// TIA Portal project "e058002v15" (V14)

(* hardware
DEVICE "S7-1200 station_1"  SIMATIC 1200-Station
   slot 0: "Rack S7-1200"  Rack  V1.0
   slot 1: "PLC_1"  CPU 1212C DC/DC/DC  6ES7 212-1AE31-0XB0  V3.0
   slot 2: "DI 8x24VDC/DQ 8xRelay_1"  SM 1223 DI8/DQ8 x relay  6ES7 223-1PH32-0XB0  V2.0
DEVICE "U9.3"  KTP600 Basic mono PN
   slot 0: "HMI"  HMI  6AV6 647-0AB11-3AX0  12.0.0.0
   slot 1: "HMI_RT_2"  KTP600 Basic mono PN  6AV6 647-0AB11-3AX0  12.0.0.0
   slot 5: "U9.3._CP_1"  Interfaz PROFINET
      slot 1: "Interfaz PROFINET_1"  Interfaz PROFINET
         slot 1: "Port_1"  Port
*)

// ===== PLC "PLC_1"  CPU 1212C DC/DC/DC =====

VAR_GLOBAL   // PLC tag table "Tabla de variables estándar"
   "System_Byte" AT %MB2 : Byte;
   "FirstScan" AT %M2.0 : Bool;
   "DiagStatusUpdate" AT %M2.1 : Bool;
   "AlwaysTRUE" AT %M2.2 : Bool;
   "AlwaysFALSE" AT %M2.3 : Bool;
   "Cuenta_Actual" AT %MW12 : Int;
   "PV_Cuenta_Rech" AT %MW14 : Int;
   "Reset_Cuenta" AT %M3.0 : Bool;
   "Aux_Ala_Enc" AT %MD220 : DInt;
   "Tag_1" AT %M231.0 : Bool;
   "Flanco falla de encoder" AT %M232.0 : Bool;
   "Tag_2" AT %M233.0 : Bool;
   "Tag_3" AT %M232.1 : Bool;
   "Flc_Ala_Encoder" AT %M234.0 : Bool;
   "Tag_4" AT %M231.2 : Bool;
   "Aux_Ala_Enc2" AT %MD224 : DInt;
   "Aux_Ala_Enc3" AT %MD240 : DInt;
   "Flc_FallaxCuentas" AT %M234.1 : Bool;
END_VAR

VAR_GLOBAL   // PLC tag table "00_Entradas"
   "iSns_PresenciaTapa" AT %I0.3 : Bool;   // S5.3 Sensor Presencia de Tapa
   "iSns_PresenciaBotella" AT %I0.2 : Bool;   // S5.4 Sensor Presencia de Botella
   "iCont_Encóder" AT %ID1000 : DInt;   // Valor Contador Encóder
   "reserva(1)" AT %I0.7 : Bool;   // Parada de emergencia caja mecanica
   "iPulsadorInicio" AT %I1.1 : Bool;   // Pulsador Inicio en caja mecanica.
   "iPulsadorParada" AT %I1.0 : Bool;   // Pulsador de parada en caja mecanica.
   "reserva" AT %I0.5 : Bool;   // Parada de emergencia en caja gris.
   "iSns_FuerzaDedos" AT %I1.2 : Bool;   // Sensor de fuerza de los dedos
END_VAR

VAR_GLOBAL   // PLC tag table "01_Salidas"
   "oRly_Pateador" AT %Q0.0 : Bool;   // R1 - Pateador
   "oRly_Embrague" AT %Q0.2 : Bool;   // R3 - Embrague
   "oLuzIndicadora" AT %Q0.4 : Bool;   // Luz indicadora de estado automatico/manual
END_VAR

VAR_GLOBAL   // PLC tag table "02_General"
   "SiempreEn_0" AT %M0.0 : Bool;   // Este Bit Siempre está en 0
   "SiempreEn_1" AT %M0.1 : Bool;   // Este Bit Siempre está en 1
   "Reset_Contador" AT %M0.2 : Bool;   // Señal para reset de contador
   "Modo" AT %M0.3 : Bool;   // Modo de funcionamiento- 0 : Parado 1: Automático
   "ParadaMaxBotRecha" AT %M0.4 : Bool;   // Parada Por Máxima cantidad de botellas rechazadas.
   "Falla_ParadaDeLinea" AT %M0.5 : Bool;   // Parada de linea por alguna falla.
   "mCont_Encoder_Anterior" AT %MD50 : DInt;
   "xFNPul_Parada" AT %M0.6 : Bool;
END_VAR

VAR_GLOBAL   // PLC tag table "03_Pateador"
   "PresenciaDeBotella" AT %M1.0 : Bool;   // Marca que indica precencia de botella.
   "PrecenciaDeBot_Y_Tapa" AT %M1.1 : Bool;   // Marca que indica precencia de tapa.
   "Botella_Sin_Tapa" AT %M1.2 : Bool;   // Marca que indica botella sin tapa
   "Ant_Botella_Sin_Tapa" AT %M1.3 : Bool;   // Valor anterior de marca que indica botella sin tapa.
   "Ord_Patear" AT %M1.4 : Bool;   // Orden para patear
   "Ant_Ord_Patear" AT %M1.5 : Bool;   // Valor anterior de orden para patear
   "Ant1_Ord_Patear" AT %M1.6 : Bool;
END_VAR

VAR_GLOBAL   // PLC tag table "05_Auxiliares"
   "AuxiliarSuma" AT %MD100 : DInt;
   "Auxiliar_1" AT %M104.0 : Bool;
   "Auxiliar_2" AT %M104.1 : Bool;
   "Auxiliar_3" AT %M104.2 : Bool;
   "Auxiliar_4" AT %M104.3 : Bool;
   "Auxiliar_5" AT %M104.4 : Bool;
   "Auxiliar_6" AT %M104.5 : Bool;
   "Auxiliar_7" AT %M104.6 : Bool;
   "Auxiliar_8" AT %M104.7 : Bool;
   "DWordTemp" AT %MD106 : DInt;
END_VAR

VAR_GLOBAL   // PLC tag table "06_Flancos"
   "fp_iSns_PresenciaTapa" AT %M10.0 : Bool;
   "fn_iSns_PresenciaTapa" AT %M10.1 : Bool;
   "fp_iSns_PresenciaBotella" AT %M10.2 : Bool;
   "fn_iSns_PresenciaBotella" AT %M10.3 : Bool;
END_VAR

VAR_GLOBAL   // PLC tag table "10_Simulacion"
   "sim_iSnsBotella" AT %M200.0 : Bool;
   "sim_iSnsTapa" AT %M200.1 : Bool;
   "sim_iPulInicio" AT %M200.2 : Bool;
   "sim_auxLoopEncoder" AT %M200.3 : Bool;
   "sim_auxFNLoop" AT %M200.4 : Bool;
END_VAR

DATA_BLOCK "100_Receta_Actual"   // DB1
TITLE = Datos Botellas
{ S7_Optimized_Access := 'TRUE' }
VERSION : 0.1
// En este bloque se almacenan todos los datos realacionado a las botellas, como ser el ancho, ancho de tapa, etc.
   VAR RETAIN
      Ancho_Max_Botella : DInt := 75;
      Cuenta_Patear : DInt := 430;
      Tiempo_Pateado : Time := T#50ms;
   END_VAR
BEGIN
END_DATA_BLOCK

DATA_BLOCK "102_Datos"   // DB2
{ S7_Optimized_Access := 'TRUE' }
VERSION : 0.1
   VAR
      Encoder_MaxCuenta : DInt := 1000000;   // Maxima cuenta del contador.
      Encoder_ValorActual : DInt;   // Variable donde alamceno valor de contador.
      Encoder_CuentaPatear : DInt;   // Valor de encoder que debe patear.
      Encoder_ValorFinBotella : DInt;   // Variable auxiliar para calculo de valor relativo del contador, sin reseteo
      NumMaxBotARechazar : Int;   // Numero maximo de botellas a rechazar, si pasa este numero genera una parada de linea.
      IndiceMaxBotARechazar : Int;   // Numero maximo del indice para rechazar botellas.
   END_VAR
BEGIN
END_DATA_BLOCK

DATA_BLOCK "101_Arreglo"   // DB4
TITLE = Arreglos
{ S7_Optimized_Access := 'TRUE' }
VERSION : 0.1
// Este bloque contiene los arreglos que se utilizan para la logica de cuenta para patear.
   VAR
      Arr_Cuenta_Patear : Array[0..9] of DInt;
      Indice : Int;
   END_VAR
BEGIN
END_DATA_BLOCK

DATA_BLOCK "103_Medición"   // DB6
{ S7_Optimized_Access := 'TRUE' }
VERSION : 0.1
   VAR
      AnchoBotellaMedicion : DInt;   // Medicion de ancho de botella
      ContadorMedicionInicio : DInt;   // Valor contador cuando ingresa botella
      ContadorMedicionFin : DInt;   // Valor contador cuando sale botella
      MedicionActivada : Bool;
      BotellaPresenteMedicion : Bool;
      MedicionRealizada : Bool;
   END_VAR
BEGIN
END_DATA_BLOCK

DATA_BLOCK "104_HMI_a_PLC"   // DB7
{ S7_Optimized_Access := 'TRUE' }
VERSION : 0.1
   VAR
      Reset : Bool;
      AnchoBotella : DInt := 75;
      CantidadPulsosPatear : DInt := 430;
      Tiempo_Pateado : Time := T#50ms;
      Cuenta_Actual : DInt;
   END_VAR
BEGIN
END_DATA_BLOCK

// folder: Alarma

DATA_BLOCK "ALA_PRE"   // DB70
{ S7_Optimized_Access := 'FALSE' }
VERSION : 0.1
   VAR
      Falla_09 : Bool;
      Falla_10 : Bool;
      Falla_11 : Bool;
      Falla_12 : Bool;
      Falla_13 : Bool;
      Falla_14 : Bool;
      Falla_15 : Bool;
      Falla_16 : Bool;
      Falla_01 : Bool;
      Falla_02 : Bool;
      Falla_03 : Bool;
      Falla_04 : Bool;
      Falla_05 : Bool;
      Falla_06 : Bool;
      Falla_07 : Bool;
      Falla_08 : Bool;
      Falla_25 : Bool;
      Falla_26 : Bool;
      Falla_27 : Bool;
      Falla_28 : Bool;
      Falla_29 : Bool;
      Falla_30 : Bool;
      Falla_31 : Bool;
      Falla_32 : Bool;
      Falla_17 : Bool;
      Falla_18 : Bool;
      Falla_19 : Bool;
      Falla_20 : Bool;
      Falla_21 : Bool;
      Falla_22 : Bool;
      Falla_23 : Bool;
      Falla_24 : Bool;
   END_VAR
BEGIN
END_DATA_BLOCK

DATA_BLOCK "ALA_MEM"   // DB71
{ S7_Optimized_Access := 'FALSE' }
VERSION : 0.1
   VAR
      Alarma_09 : Bool;
      Alarma_10 : Bool;
      Alarma_11 : Bool;
      Alarma_12 : Bool;
      Alarma_13 : Bool;
      Alarma_14 : Bool;
      Alarma_15 : Bool;
      Alarma_16 : Bool;
      Alarma_01 : Bool;
      Alarma_02 : Bool;
      Alarma_03 : Bool;
      Alarma_04 : Bool;
      Alarma_05 : Bool;
      Alarma_06 : Bool;
      Alarma_07 : Bool;
      Alarma_08 : Bool;
      Alarma_25 : Bool;
      Alarma_26 : Bool;
      Alarma_27 : Bool;
      Alarma_28 : Bool;
      Alarma_29 : Bool;
      Alarma_30 : Bool;
      Alarma_31 : Bool;
      Alarma_32 : Bool;
      Alarma_17 : Bool;
      Alarma_18 : Bool;
      Alarma_19 : Bool;
      Alarma_20 : Bool;
      Alarma_21 : Bool;
      Alarma_22 : Bool;
      Alarma_23 : Bool;
      Alarma_24 : Bool;
   END_VAR
BEGIN
END_DATA_BLOCK

DATA_BLOCK "ALA_REC"   // DB72
{ S7_Optimized_Access := 'FALSE' }
VERSION : 0.1
   VAR
      Ala_Rec_09 : Bool;
      Ala_Rec_10 : Bool;
      Ala_Rec_11 : Bool;
      Ala_Rec_12 : Bool;
      Ala_Rec_13 : Bool;
      Ala_Rec_14 : Bool;
      Ala_Rec_15 : Bool;
      Ala_Rec_16 : Bool;
      Ala_Rec_01 : Bool;
      Ala_Rec_02 : Bool;
      Ala_Rec_03 : Bool;
      Ala_Rec_04 : Bool;
      Ala_Rec_05 : Bool;
      Ala_Rec_06 : Bool;
      Ala_Rec_07 : Bool;
      Ala_Rec_08 : Bool;
      Ala_Rec_25 : Bool;
      Ala_Rec_26 : Bool;
      Ala_Rec_27 : Bool;
      Ala_Rec_28 : Bool;
      Ala_Rec_29 : Bool;
      Ala_Rec_30 : Bool;
      Ala_Rec_31 : Bool;
      Ala_Rec_32 : Bool;
      Ala_Rec_17 : Bool;
      Ala_Rec_18 : Bool;
      Ala_Rec_19 : Bool;
      Ala_Rec_20 : Bool;
      Ala_Rec_21 : Bool;
      Ala_Rec_22 : Bool;
      Ala_Rec_23 : Bool;
      Ala_Rec_24 : Bool;
   END_VAR
BEGIN
END_DATA_BLOCK

// folder: System blocks/Program resources

DATA_BLOCK "IEC_Timer_0_DB"   // DB5
{ S7_Optimized_Access := 'TRUE' }
AUTHOR : Simatic
FAMILY : IEC
NAME : IEC_TMR
VERSION : 1.0
// stored: InstanceOfName IEC_TIMER
"IEC_TIMER"
BEGIN
END_DATA_BLOCK

DATA_BLOCK "sim_tonLoopEncoder"   // DB8
{ S7_Optimized_Access := 'TRUE' }
AUTHOR : Simatic
FAMILY : IEC
NAME : IEC_TMR
VERSION : 1.0
// stored: InstanceOfName IEC_TIMER
"IEC_TIMER"
BEGIN
END_DATA_BLOCK

DATA_BLOCK "Temp_Parada_Cinta"   // DB9
{ S7_Optimized_Access := 'TRUE' }
AUTHOR : Simatic
FAMILY : IEC
NAME : IEC_TMR
VERSION : 1.0
// stored: InstanceOfName IEC_TIMER
"IEC_TIMER"
BEGIN
END_DATA_BLOCK

DATA_BLOCK "Bot_Rechazada"   // DB10
{ S7_Optimized_Access := 'TRUE' }
AUTHOR : Simatic
FAMILY : IEC
NAME : CNTR
VERSION : 1.0
// stored: InstanceOfName IEC_COUNTER
"IEC_COUNTER"
BEGIN
END_DATA_BLOCK

DATA_BLOCK "IEC_Timer_0_DB_1"   // DB11
{ S7_Optimized_Access := 'TRUE' }
AUTHOR : Simatic
FAMILY : IEC
NAME : IEC_TMR
VERSION : 1.0
// stored: InstanceOfName IEC_TIMER
"IEC_TIMER"
BEGIN
END_DATA_BLOCK

DATA_BLOCK "IEC_Timer_0_DB_2"   // DB12
{ S7_Optimized_Access := 'TRUE' }
AUTHOR : Simatic
FAMILY : IEC
NAME : IEC_TMR
VERSION : 1.0
// stored: InstanceOfName IEC_TIMER
"IEC_TIMER"
BEGIN
END_DATA_BLOCK

// folder: (top level)

FUNCTION "04_Pateador" : Void   // FC1, LAD
TITLE = Lógica del Pateador
{ S7_Optimized_Access := 'TRUE' }
VERSION : 0.1
// En este bloque se resuelve toda la lógica necesaria para activar el pateador.
   VAR_TEMP
      dist_Bot_a_pat : DInt;
   END_VAR
   VAR_TEMP   // added for the SCL form of the ladder/FBD networks
      _w1 : Bool;
      _w2 : Bool;
   END_VAR
BEGIN

REGION Network 1: Reset de contador.
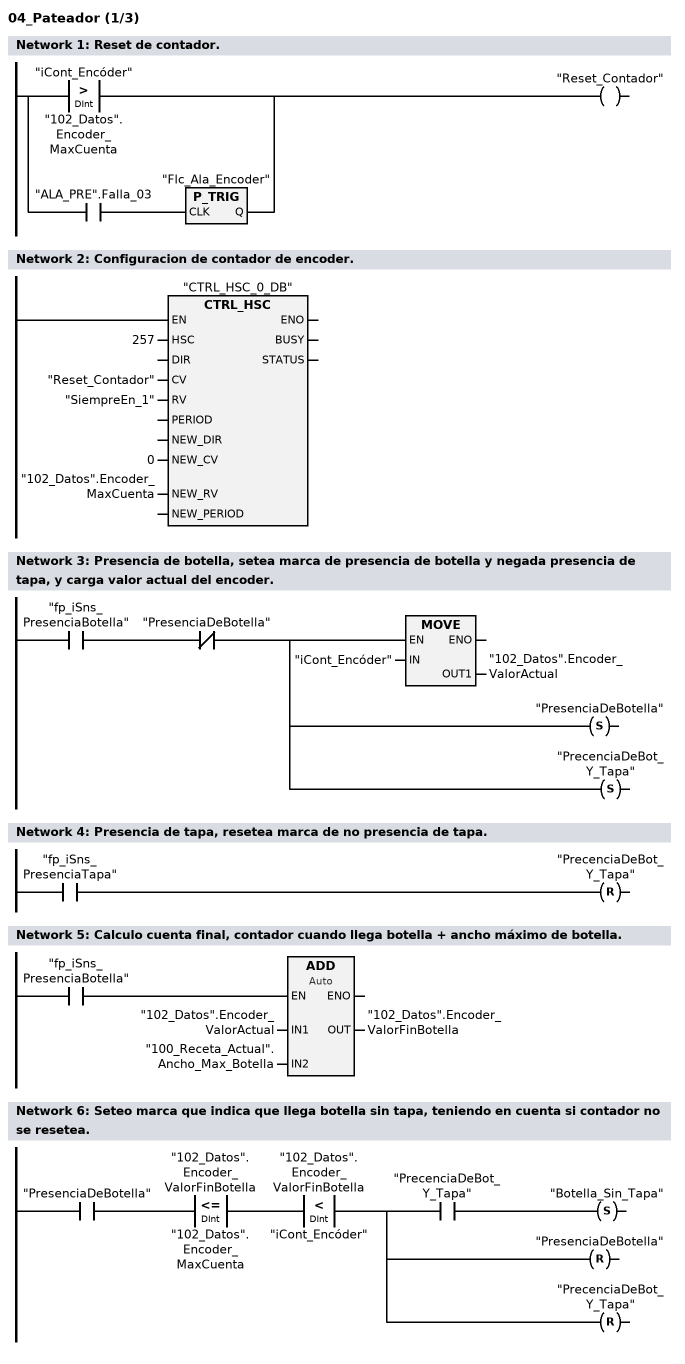
   RUNG wire#powerrail
      { S7_Templates := "SrcType := DInt" } GT_Contact(in1 := "iCont_Encóder", in2 := "102_Datos".Encoder_MaxCuenta)
      wire#w1
      Coil( "Reset_Contador" )
   END_RUNG
   RUNG wire#powerrail
      Contact( "ALA_PRE".Falla_03 )
      P_Trig( "Flc_Ala_Encoder" )
   END_RUNG wire#w1
   // the same network as SCL:
   #_w1 := "ALA_PRE".Falla_03 AND NOT "Flc_Ala_Encoder";   // rising edge
   "Flc_Ala_Encoder" := "ALA_PRE".Falla_03;
   "Reset_Contador" := ("iCont_Encóder" > "102_Datos".Encoder_MaxCuenta) OR #_w1;
END_REGION

REGION Network 2: Configuracion de contador de encoder.
   "CTRL_HSC_0_DB"(HSC := 257,   // CTRL_HSC
                   CV := "Reset_Contador",
                   RV := "SiempreEn_1",
                   NEW_CV := 0,
                   NEW_RV := "102_Datos".Encoder_MaxCuenta);
END_REGION

REGION Network 3: Presencia de botella, setea marca de presencia de botella y negada presencia de tapa, y carga valor actual del encoder.
   RUNG wire#powerrail
      Contact( "fp_iSns_PresenciaBotella" )
      I_Contact( "PresenciaDeBotella" )
      wire#w1
      { S7_GenerateENO := "TRUE" } Move(in := "iCont_Encóder", out1 => "102_Datos".Encoder_ValorActual)
   END_RUNG
   RUNG wire#w1
      S_Coil( "PresenciaDeBotella" )
   END_RUNG
   RUNG wire#w1
      S_Coil( "PrecenciaDeBot_Y_Tapa" )
   END_RUNG
   // the same network as SCL:
   IF "fp_iSns_PresenciaBotella" AND NOT "PresenciaDeBotella" THEN
       "102_Datos".Encoder_ValorActual := "iCont_Encóder";
   END_IF;
   #_w1 := "fp_iSns_PresenciaBotella" AND NOT "PresenciaDeBotella";
   IF #_w1 THEN
       "PresenciaDeBotella" := TRUE;
       "PrecenciaDeBot_Y_Tapa" := TRUE;
   END_IF;
END_REGION

REGION Network 4: Presencia de tapa, resetea marca de no presencia de tapa.
   RUNG wire#powerrail
      Contact( "fp_iSns_PresenciaTapa" )
      R_Coil( "PrecenciaDeBot_Y_Tapa" )
   END_RUNG
   // the same network as SCL:
   IF "fp_iSns_PresenciaTapa" THEN "PrecenciaDeBot_Y_Tapa" := FALSE; END_IF;
END_REGION

REGION Network 5: Calculo cuenta final, contador cuando llega botella + ancho máximo de botella.
   RUNG wire#powerrail
      Contact( "fp_iSns_PresenciaBotella" )
      { S7_GenerateENO := "TRUE" } Add(in1 := "102_Datos".Encoder_ValorActual, in2 := "100_Receta_Actual".Ancho_Max_Botella, out => "102_Datos".Encoder_ValorFinBotella)
   END_RUNG
   // the same network as SCL:
   IF "fp_iSns_PresenciaBotella" THEN
       "102_Datos".Encoder_ValorFinBotella := "102_Datos".Encoder_ValorActual + "100_Receta_Actual".Ancho_Max_Botella;
   END_IF;
END_REGION

REGION Network 6: Seteo marca que indica que llega botella sin tapa, teniendo en cuenta si contador no se resetea.
   RUNG wire#powerrail
      Contact( "PresenciaDeBotella" )
      { S7_Templates := "SrcType := DInt" } LE_Contact(in1 := "102_Datos".Encoder_ValorFinBotella, in2 := "102_Datos".Encoder_MaxCuenta)
      { S7_Templates := "SrcType := DInt" } LT_Contact(in1 := "102_Datos".Encoder_ValorFinBotella, in2 := "iCont_Encóder")
      wire#w1
      Contact( "PrecenciaDeBot_Y_Tapa" )
      S_Coil( "Botella_Sin_Tapa" )
   END_RUNG
   RUNG wire#w1
      R_Coil( "PresenciaDeBotella" )
   END_RUNG
   RUNG wire#w1
      R_Coil( "PrecenciaDeBot_Y_Tapa" )
   END_RUNG
   // the same network as SCL:
   #_w1 := "PresenciaDeBotella" AND ("102_Datos".Encoder_ValorFinBotella <= "102_Datos".Encoder_MaxCuenta) AND ("102_Datos".Encoder_ValorFinBotella < "iCont_Encóder");
   IF #_w1 AND "PrecenciaDeBot_Y_Tapa" THEN "Botella_Sin_Tapa" := TRUE; END_IF;
   IF #_w1 THEN
       "PresenciaDeBotella" := FALSE;
       "PrecenciaDeBot_Y_Tapa" := FALSE;
   END_IF;
END_REGION

REGION Network 7: Seteo marca que indica que llega botella sin tapa, teniendo en cuenta el caso que el contador se resetea.
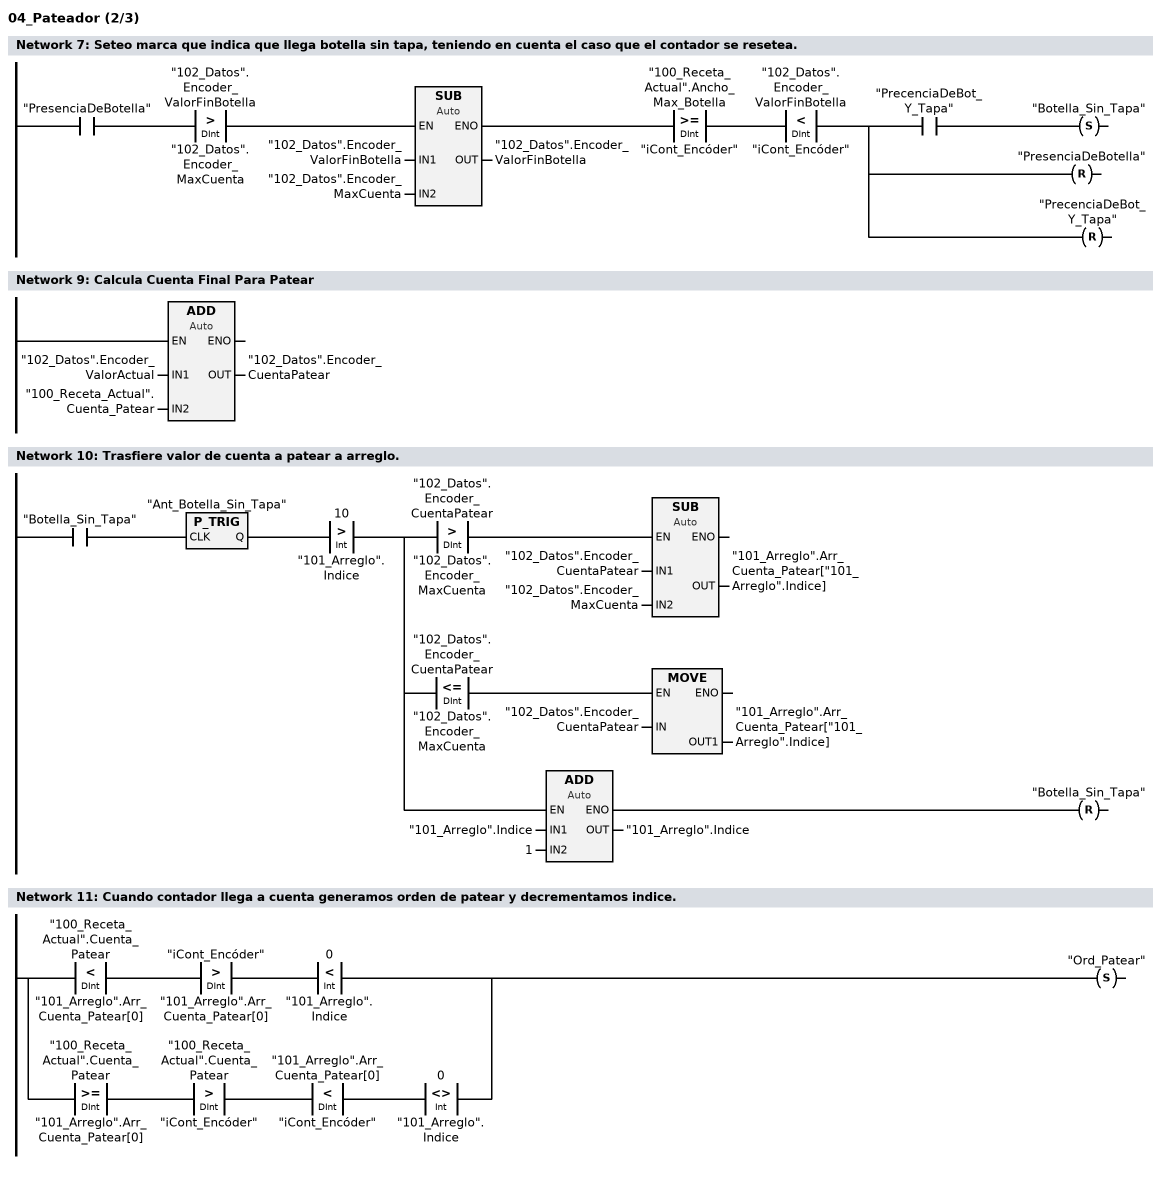
   RUNG wire#powerrail
      Contact( "PresenciaDeBotella" )
      { S7_Templates := "SrcType := DInt" } GT_Contact(in1 := "102_Datos".Encoder_ValorFinBotella, in2 := "102_Datos".Encoder_MaxCuenta)
      { S7_GenerateENO := "TRUE" } Sub(in1 := "102_Datos".Encoder_ValorFinBotella, in2 := "102_Datos".Encoder_MaxCuenta, out => "102_Datos".Encoder_ValorFinBotella)
      { S7_Templates := "SrcType := DInt" } GE_Contact(in1 := "100_Receta_Actual".Ancho_Max_Botella, in2 := "iCont_Encóder")
      { S7_Templates := "SrcType := DInt" } LT_Contact(in1 := "102_Datos".Encoder_ValorFinBotella, in2 := "iCont_Encóder")
      wire#w1
      Contact( "PrecenciaDeBot_Y_Tapa" )
      S_Coil( "Botella_Sin_Tapa" )
   END_RUNG
   RUNG wire#w1
      R_Coil( "PresenciaDeBotella" )
   END_RUNG
   RUNG wire#w1
      R_Coil( "PrecenciaDeBot_Y_Tapa" )
   END_RUNG
   // the same network as SCL:
   // ENO of a box is taken as its EN; it also drops when the box reports an error
   #_w1 := "PresenciaDeBotella" AND ("102_Datos".Encoder_ValorFinBotella > "102_Datos".Encoder_MaxCuenta);
   IF #_w1 THEN
       "102_Datos".Encoder_ValorFinBotella := "102_Datos".Encoder_ValorFinBotella - "102_Datos".Encoder_MaxCuenta;
   END_IF;
   #_w2 := #_w1 AND ("100_Receta_Actual".Ancho_Max_Botella >= "iCont_Encóder") AND ("102_Datos".Encoder_ValorFinBotella < "iCont_Encóder");
   IF #_w2 AND "PrecenciaDeBot_Y_Tapa" THEN "Botella_Sin_Tapa" := TRUE; END_IF;
   IF #_w2 THEN
       "PresenciaDeBotella" := FALSE;
       "PrecenciaDeBot_Y_Tapa" := FALSE;
   END_IF;
END_REGION

REGION Network 8: Marca que indica precencia de botella.
END_REGION

REGION Network 9: Calcula Cuenta Final Para Patear
   RUNG wire#powerrail
      { S7_GenerateENO := "TRUE" } Add(in1 := "102_Datos".Encoder_ValorActual, in2 := "100_Receta_Actual".Cuenta_Patear, out => "102_Datos".Encoder_CuentaPatear)
   END_RUNG
   // the same network as SCL:
   "102_Datos".Encoder_CuentaPatear := "102_Datos".Encoder_ValorActual + "100_Receta_Actual".Cuenta_Patear;
END_REGION

REGION Network 10: Trasfiere valor de cuenta a patear a arreglo.
   RUNG wire#powerrail
      Contact( "Botella_Sin_Tapa" )
      P_Trig( "Ant_Botella_Sin_Tapa" )
      { S7_Templates := "SrcType := Int" } GT_Contact(in1 := 10, in2 := "101_Arreglo".Indice)
      wire#w1
      { S7_Templates := "SrcType := DInt" } GT_Contact(in1 := "102_Datos".Encoder_CuentaPatear, in2 := "102_Datos".Encoder_MaxCuenta)
      { S7_GenerateENO := "TRUE" } Sub(in1 := "102_Datos".Encoder_CuentaPatear, in2 := "102_Datos".Encoder_MaxCuenta, out => "101_Arreglo".Arr_Cuenta_Patear["101_Arreglo".Indice])
   END_RUNG
   RUNG wire#w1
      { S7_Templates := "SrcType := DInt" } LE_Contact(in1 := "102_Datos".Encoder_CuentaPatear, in2 := "102_Datos".Encoder_MaxCuenta)
      { S7_GenerateENO := "TRUE" } Move(in := "102_Datos".Encoder_CuentaPatear, out1 => "101_Arreglo".Arr_Cuenta_Patear["101_Arreglo".Indice])
   END_RUNG
   RUNG wire#w1
      { S7_GenerateENO := "TRUE" } Add(in1 := "101_Arreglo".Indice, in2 := 1, out => "101_Arreglo".Indice)
      R_Coil( "Botella_Sin_Tapa" )
   END_RUNG
   // the same network as SCL:
   // ENO of a box is taken as its EN; it also drops when the box reports an error
   #_w1 := "Botella_Sin_Tapa" AND NOT "Ant_Botella_Sin_Tapa";   // rising edge
   "Ant_Botella_Sin_Tapa" := "Botella_Sin_Tapa";
   #_w2 := #_w1 AND (10 > "101_Arreglo".Indice);
   IF #_w2 AND ("102_Datos".Encoder_CuentaPatear > "102_Datos".Encoder_MaxCuenta) THEN
       "101_Arreglo".Arr_Cuenta_Patear["101_Arreglo".Indice] := "102_Datos".Encoder_CuentaPatear - "102_Datos".Encoder_MaxCuenta;
   END_IF;
   IF #_w2 AND ("102_Datos".Encoder_CuentaPatear <= "102_Datos".Encoder_MaxCuenta) THEN
       "101_Arreglo".Arr_Cuenta_Patear["101_Arreglo".Indice] := "102_Datos".Encoder_CuentaPatear;
   END_IF;
   IF #_w2 THEN
       "101_Arreglo".Indice := "101_Arreglo".Indice + 1;
       "Botella_Sin_Tapa" := FALSE;
   END_IF;
END_REGION

REGION Network 11: Cuando contador llega a cuenta generamos orden de patear y decrementamos indice.
   RUNG wire#powerrail
      { S7_Templates := "SrcType := DInt" } LT_Contact(in1 := "100_Receta_Actual".Cuenta_Patear, in2 := "101_Arreglo".Arr_Cuenta_Patear[0])
      { S7_Templates := "SrcType := DInt" } GT_Contact(in1 := "iCont_Encóder", in2 := "101_Arreglo".Arr_Cuenta_Patear[0])
      { S7_Templates := "SrcType := Int" } LT_Contact(in1 := 0, in2 := "101_Arreglo".Indice)
      wire#w1
      S_Coil( "Ord_Patear" )
   END_RUNG
   RUNG wire#powerrail
      { S7_Templates := "SrcType := DInt" } GE_Contact(in1 := "100_Receta_Actual".Cuenta_Patear, in2 := "101_Arreglo".Arr_Cuenta_Patear[0])
      { S7_Templates := "SrcType := DInt" } GT_Contact(in1 := "100_Receta_Actual".Cuenta_Patear, in2 := "iCont_Encóder")
      { S7_Templates := "SrcType := DInt" } LT_Contact(in1 := "101_Arreglo".Arr_Cuenta_Patear[0], in2 := "iCont_Encóder")
      { S7_Templates := "SrcType := Int" } NE_Contact(in1 := 0, in2 := "101_Arreglo".Indice)
   END_RUNG wire#w1
   // the same network as SCL:
   IF (("100_Receta_Actual".Cuenta_Patear < "101_Arreglo".Arr_Cuenta_Patear[0]) AND ("iCont_Encóder" > "101_Arreglo".Arr_Cuenta_Patear[0]) AND (0 < "101_Arreglo".Indice)) OR (("100_Receta_Actual".Cuenta_Patear >= "101_Arreglo".Arr_Cuenta_Patear[0]) AND ("100_Receta_Actual".Cuenta_Patear > "iCont_Encóder") AND ("101_Arreglo".Arr_Cuenta_Patear[0] < "iCont_Encóder") AND (0 <> "101_Arreglo".Indice)) THEN
       "Ord_Patear" := TRUE;
   END_IF;
END_REGION

REGION Network 12: Correr Arreglo En una Valor de 1 a 0 y activo salida por un timepo determinado y decrementa indice
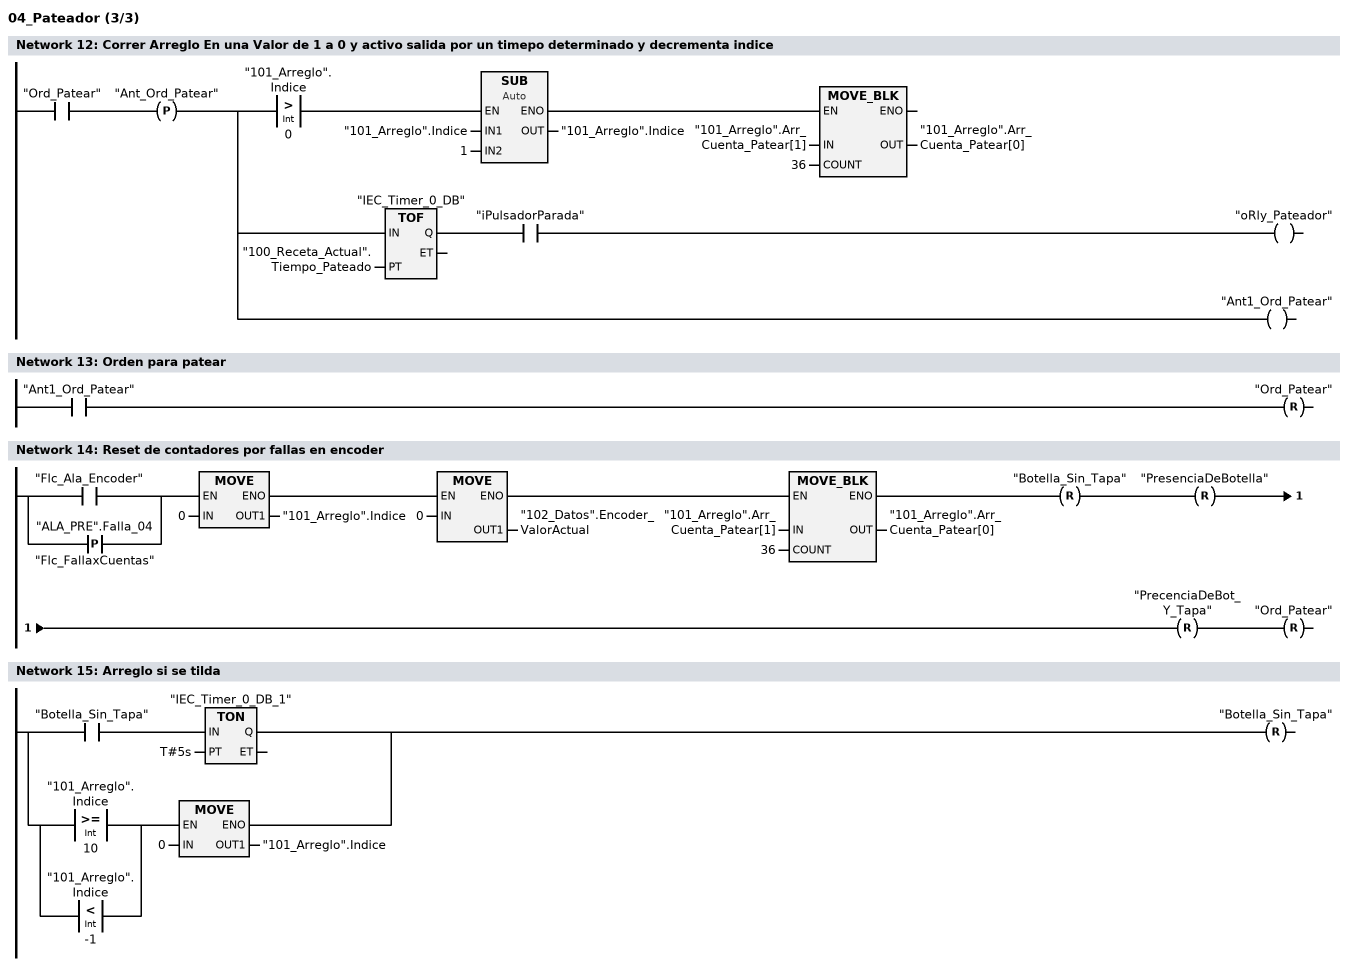
   // ENO of a box is taken as its EN; it also drops when the box reports an error
   #_w1 := "Ord_Patear" AND NOT "Ant_Ord_Patear";   // rising edge
   "Ant_Ord_Patear" := "Ord_Patear";
   #_w2 := #_w1 AND ("101_Arreglo".Indice > 0);
   IF #_w2 THEN
       "101_Arreglo".Indice := "101_Arreglo".Indice - 1;
       MOVE_BLK(IN := "101_Arreglo".Arr_Cuenta_Patear[1], COUNT := 36, OUT => "101_Arreglo".Arr_Cuenta_Patear[0]);
   END_IF;
   "IEC_Timer_0_DB".TOF(IN := #_w1, PT := "100_Receta_Actual".Tiempo_Pateado);
   "oRly_Pateador" := "IEC_Timer_0_DB".Q AND "iPulsadorParada";
   "Ant1_Ord_Patear" := #_w1;
END_REGION

REGION Network 13: Orden para patear
   RUNG wire#powerrail
      Contact( "Ant1_Ord_Patear" )
      R_Coil( "Ord_Patear" )
   END_RUNG
   // the same network as SCL:
   IF "Ant1_Ord_Patear" THEN "Ord_Patear" := FALSE; END_IF;
END_REGION

REGION Network 14: Reset de contadores por fallas en encoder
   // ENO of a box is taken as its EN; it also drops when the box reports an error
   #_w1 := "ALA_PRE".Falla_04 AND NOT "Flc_FallaxCuentas";   // rising edge of "ALA_PRE".Falla_04
   "Flc_FallaxCuentas" := "ALA_PRE".Falla_04;
   IF "Flc_Ala_Encoder" OR #_w1 THEN
       "101_Arreglo".Indice := 0;
       "102_Datos".Encoder_ValorActual := 0;
   END_IF;
   #_w2 := "Flc_Ala_Encoder" OR #_w1;
   IF #_w2 THEN
       MOVE_BLK(IN := "101_Arreglo".Arr_Cuenta_Patear[1], COUNT := 36, OUT => "101_Arreglo".Arr_Cuenta_Patear[0]);
       "Botella_Sin_Tapa" := FALSE;
       "PresenciaDeBotella" := FALSE;
       "PrecenciaDeBot_Y_Tapa" := FALSE;
       "Ord_Patear" := FALSE;
   END_IF;
END_REGION

REGION Network 15: Arreglo si se tilda
   // ENO of a box is taken as its EN; it also drops when the box reports an error
   "IEC_Timer_0_DB_1".TON(IN := "Botella_Sin_Tapa", PT := T#5s);
   #_w1 := ("101_Arreglo".Indice >= 10) OR ("101_Arreglo".Indice < (-1));
   IF #_w1 THEN "101_Arreglo".Indice := 0; END_IF;
   IF "IEC_Timer_0_DB_1".Q OR #_w1 THEN "Botella_Sin_Tapa" := FALSE; END_IF;
END_REGION
END_FUNCTION

FUNCTION "03_Medicion" : Void   // FC2, LAD
TITLE = Medicion
{ S7_Optimized_Access := 'TRUE' }
VERSION : 0.1
// En este bloque realizamos la medicion del ancho de la botella.
   VAR_TEMP   // added for the SCL form of the ladder/FBD networks
      _w1 : Bool;
   END_VAR
BEGIN

REGION Network 1: Guardamos valor de contador cuando llega botella.
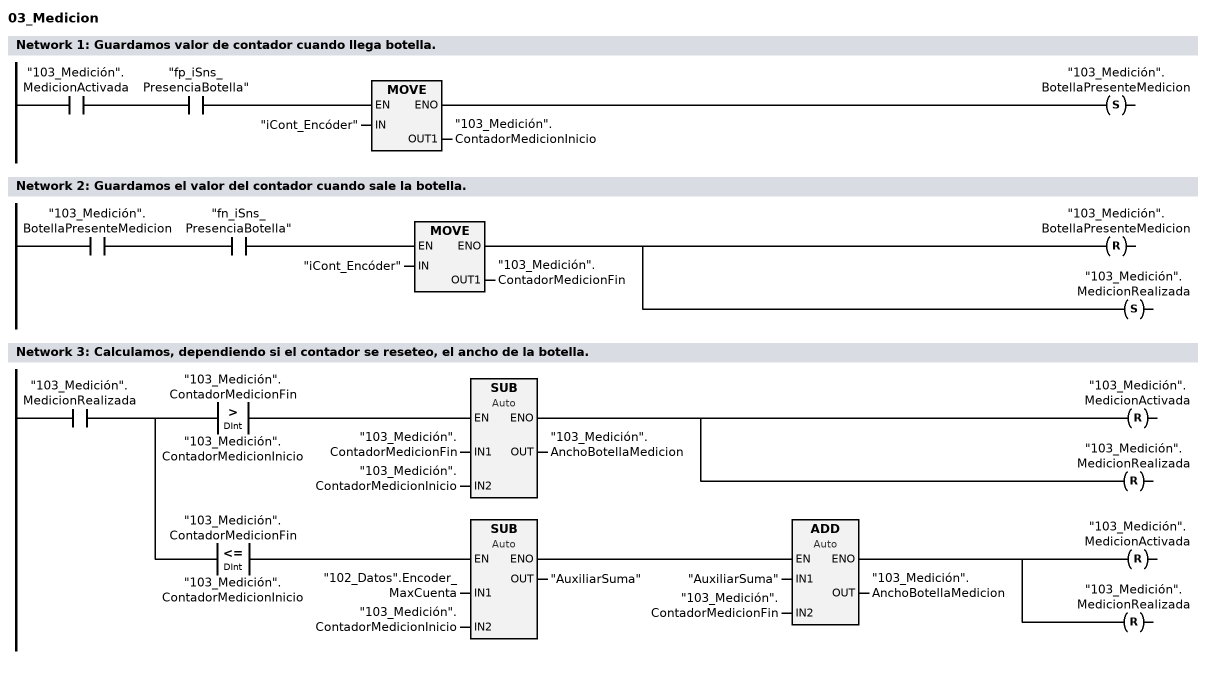
   RUNG wire#powerrail
      Contact( "103_Medición".MedicionActivada )
      Contact( "fp_iSns_PresenciaBotella" )
      { S7_GenerateENO := "TRUE" } Move(in := "iCont_Encóder", out1 => "103_Medición".ContadorMedicionInicio)
      S_Coil( "103_Medición".BotellaPresenteMedicion )
   END_RUNG
   // the same network as SCL:
   // ENO of a box is taken as its EN; it also drops when the box reports an error
   IF "103_Medición".MedicionActivada AND "fp_iSns_PresenciaBotella" THEN
       "103_Medición".ContadorMedicionInicio := "iCont_Encóder";
       "103_Medición".BotellaPresenteMedicion := TRUE;
   END_IF;
END_REGION

REGION Network 2: Guardamos el valor del contador cuando sale la botella.
   RUNG wire#powerrail
      Contact( "103_Medición".BotellaPresenteMedicion )
      Contact( "fn_iSns_PresenciaBotella" )
      { S7_GenerateENO := "TRUE" } Move(in := "iCont_Encóder", out1 => "103_Medición".ContadorMedicionFin)
      wire#w1
      R_Coil( "103_Medición".BotellaPresenteMedicion )
   END_RUNG
   RUNG wire#w1
      S_Coil( "103_Medición".MedicionRealizada )
   END_RUNG
   // the same network as SCL:
   // ENO of a box is taken as its EN; it also drops when the box reports an error
   IF "103_Medición".BotellaPresenteMedicion AND "fn_iSns_PresenciaBotella" THEN
       "103_Medición".ContadorMedicionFin := "iCont_Encóder";
   END_IF;
   #_w1 := "103_Medición".BotellaPresenteMedicion AND "fn_iSns_PresenciaBotella";
   IF #_w1 THEN
       "103_Medición".BotellaPresenteMedicion := FALSE;
       "103_Medición".MedicionRealizada := TRUE;
   END_IF;
END_REGION

REGION Network 3: Calculamos, dependiendo si el contador se reseteo, el ancho de la botella.
   RUNG wire#powerrail
      Contact( "103_Medición".MedicionRealizada )
      wire#w1
      { S7_Templates := "SrcType := DInt" } GT_Contact(in1 := "103_Medición".ContadorMedicionFin, in2 := "103_Medición".ContadorMedicionInicio)
      { S7_GenerateENO := "TRUE" } Sub(in1 := "103_Medición".ContadorMedicionFin, in2 := "103_Medición".ContadorMedicionInicio, out => "103_Medición".AnchoBotellaMedicion)
      wire#w2
      R_Coil( "103_Medición".MedicionActivada )
   END_RUNG
   RUNG wire#w2
      R_Coil( "103_Medición".MedicionRealizada )
   END_RUNG
   RUNG wire#w1
      { S7_Templates := "SrcType := DInt" } LE_Contact(in1 := "103_Medición".ContadorMedicionFin, in2 := "103_Medición".ContadorMedicionInicio)
      { S7_GenerateENO := "TRUE" } Sub(in1 := "102_Datos".Encoder_MaxCuenta, in2 := "103_Medición".ContadorMedicionInicio, out => "AuxiliarSuma")
      { S7_GenerateENO := "TRUE" } Add(in1 := "AuxiliarSuma", in2 := "103_Medición".ContadorMedicionFin, out => "103_Medición".AnchoBotellaMedicion)
      wire#w3
      R_Coil( "103_Medición".MedicionActivada )
   END_RUNG
   RUNG wire#w3
      R_Coil( "103_Medición".MedicionRealizada )
   END_RUNG
   // the same network as SCL:
   // ENO of a box is taken as its EN; it also drops when the box reports an error
   IF "103_Medición".MedicionRealizada AND ("103_Medición".ContadorMedicionFin > "103_Medición".ContadorMedicionInicio) THEN
       "103_Medición".AnchoBotellaMedicion := "103_Medición".ContadorMedicionFin - "103_Medición".ContadorMedicionInicio;
       "103_Medición".MedicionActivada := FALSE;
   END_IF;
   #_w1 := "103_Medición".MedicionRealizada;
   IF "103_Medición".MedicionRealizada AND ("103_Medición".ContadorMedicionFin > "103_Medición".ContadorMedicionInicio) THEN
       "103_Medición".MedicionRealizada := FALSE;
   END_IF;
   IF #_w1 AND ("103_Medición".ContadorMedicionFin <= "103_Medición".ContadorMedicionInicio) THEN
       "AuxiliarSuma" := "102_Datos".Encoder_MaxCuenta - "103_Medición".ContadorMedicionInicio;
       "103_Medición".AnchoBotellaMedicion := "AuxiliarSuma" + "103_Medición".ContadorMedicionFin;
       "103_Medición".MedicionActivada := FALSE;
       "103_Medición".MedicionRealizada := FALSE;
   END_IF;
END_REGION
END_FUNCTION

FUNCTION "00_Alarmas" : Void   // FC3, LAD
{ S7_Optimized_Access := 'TRUE' }
VERSION : 0.1
   VAR_TEMP
      dist_Bot_a_pat : DInt;
   END_VAR
   VAR_TEMP   // added for the SCL form of the ladder/FBD networks
      _w1 : Bool;
   END_VAR
BEGIN

REGION Network 1: Parada manual. Emergencia o Stop del embrague del pateador.
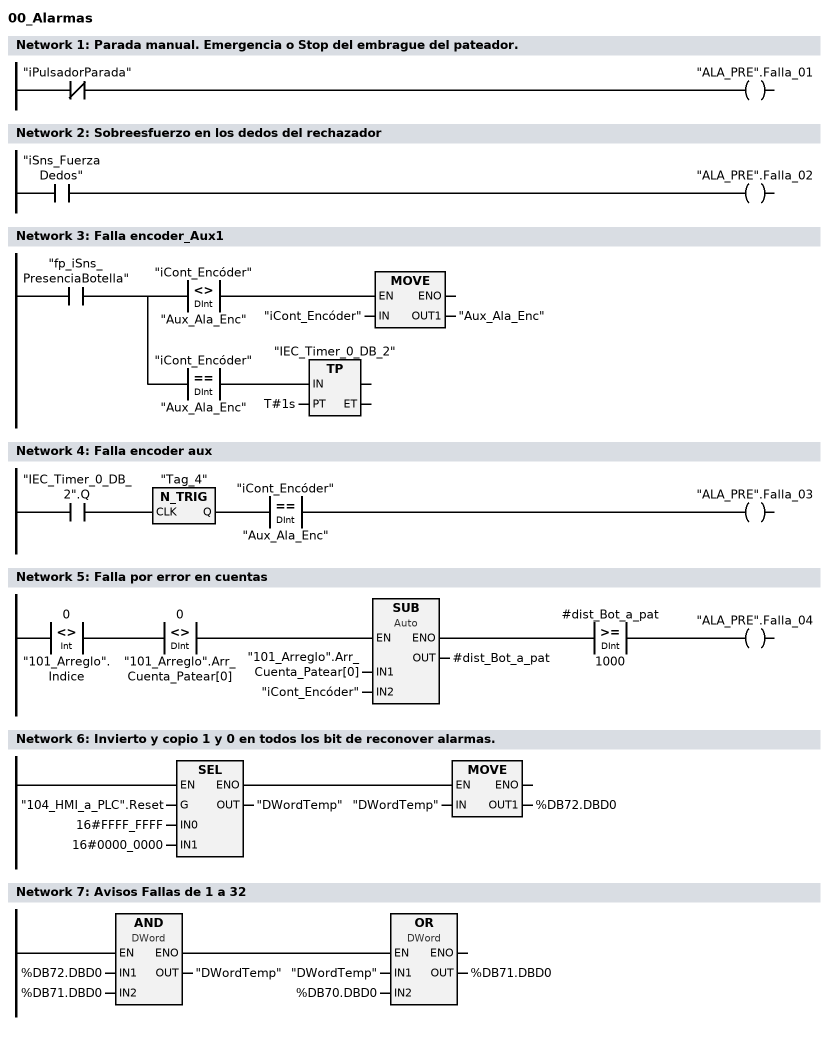
   RUNG wire#powerrail
      I_Contact( "iPulsadorParada" )
      Coil( "ALA_PRE".Falla_01 )
   END_RUNG
   // the same network as SCL:
   "ALA_PRE".Falla_01 := NOT "iPulsadorParada";
END_REGION

REGION Network 2: Sobreesfuerzo en los dedos del rechazador
   RUNG wire#powerrail
      Contact( "iSns_FuerzaDedos" )
      Coil( "ALA_PRE".Falla_02 )
   END_RUNG
   // the same network as SCL:
   "ALA_PRE".Falla_02 := "iSns_FuerzaDedos";
END_REGION

REGION Network 3: Falla encoder_Aux1
   IF "fp_iSns_PresenciaBotella" AND ("iCont_Encóder" <> "Aux_Ala_Enc") THEN
       "Aux_Ala_Enc" := "iCont_Encóder";
   END_IF;
   "IEC_Timer_0_DB_2".TP(IN := "fp_iSns_PresenciaBotella" AND ("iCont_Encóder" = "Aux_Ala_Enc"), PT := T#1s);
END_REGION

REGION Network 4: Falla encoder aux
   RUNG wire#powerrail
      Contact( "IEC_Timer_0_DB_2".Q )
      N_Trig( "Tag_4" )
      { S7_Templates := "SrcType := DInt" } EQ_Contact(in1 := "iCont_Encóder", in2 := "Aux_Ala_Enc")
      Coil( "ALA_PRE".Falla_03 )
   END_RUNG
   // the same network as SCL:
   #_w1 := NOT "IEC_Timer_0_DB_2".Q AND "Tag_4";   // falling edge
   "Tag_4" := "IEC_Timer_0_DB_2".Q;
   "ALA_PRE".Falla_03 := #_w1 AND ("iCont_Encóder" = "Aux_Ala_Enc");
END_REGION

REGION Network 5: Falla por error en cuentas
   RUNG wire#powerrail
      { S7_Templates := "SrcType := Int" } NE_Contact(in1 := 0, in2 := "101_Arreglo".Indice)
      { S7_Templates := "SrcType := DInt" } NE_Contact(in1 := 0, in2 := "101_Arreglo".Arr_Cuenta_Patear[0])
      { S7_GenerateENO := "TRUE" } Sub(in1 := "101_Arreglo".Arr_Cuenta_Patear[0], in2 := "iCont_Encóder", out => #dist_Bot_a_pat)
      { S7_Templates := "SrcType := DInt" } GE_Contact(in1 := #dist_Bot_a_pat, in2 := 1000)
      Coil( "ALA_PRE".Falla_04 )
   END_RUNG
   // the same network as SCL:
   // ENO of a box is taken as its EN; it also drops when the box reports an error
   #_w1 := (0 <> "101_Arreglo".Indice) AND (0 <> "101_Arreglo".Arr_Cuenta_Patear[0]);
   IF #_w1 THEN #dist_Bot_a_pat := "101_Arreglo".Arr_Cuenta_Patear[0] - "iCont_Encóder"; END_IF;
   "ALA_PRE".Falla_04 := #_w1 AND (#dist_Bot_a_pat >= 1000);
END_REGION

REGION Network 6: Invierto y copio 1 y 0 en todos los bit de reconover alarmas.
   // ENO of a box is taken as its EN; it also drops when the box reports an error
   "DWordTemp" := SEL(G := "104_HMI_a_PLC".Reset, IN0 := 16#FFFF_FFFF, IN1 := 16#0000_0000);
   %DB72.DBD0 := "DWordTemp";
END_REGION

REGION Network 7: Avisos Fallas de 1 a 32
   // no checked SCL form for this network; see the picture
END_REGION
END_FUNCTION

FUNCTION "01_General" : Void   // FC4, LAD
{ S7_Optimized_Access := 'TRUE' }
VERSION : 0.1
BEGIN

REGION Network 1: Set modo automatico
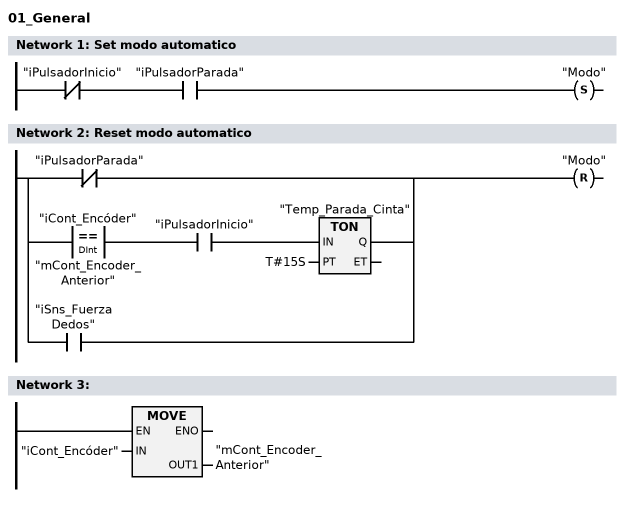
   RUNG wire#powerrail
      I_Contact( "iPulsadorInicio" )
      Contact( "iPulsadorParada" )
      S_Coil( "Modo" )
   END_RUNG
   // the same network as SCL:
   IF NOT "iPulsadorInicio" AND "iPulsadorParada" THEN "Modo" := TRUE; END_IF;
END_REGION

REGION Network 2: Reset modo automatico
   "Temp_Parada_Cinta".TON(IN := ("iCont_Encóder" = "mCont_Encoder_Anterior") AND "iPulsadorInicio",
                           PT := T#15S);
   IF NOT "iPulsadorParada" OR "Temp_Parada_Cinta".Q OR "iSns_FuerzaDedos" THEN "Modo" := FALSE; END_IF;
END_REGION

REGION Network 3
   RUNG wire#powerrail
      { S7_GenerateENO := "TRUE" } Move(in := "iCont_Encóder", out1 => "mCont_Encoder_Anterior")
   END_RUNG
   // the same network as SCL:
   "mCont_Encoder_Anterior" := "iCont_Encóder";
END_REGION
END_FUNCTION

FUNCTION "06_Salidas" : Void   // FC5, LAD
{ S7_Optimized_Access := 'TRUE' }
VERSION : 0.1
BEGIN

REGION Network 1: R3 - Embrague
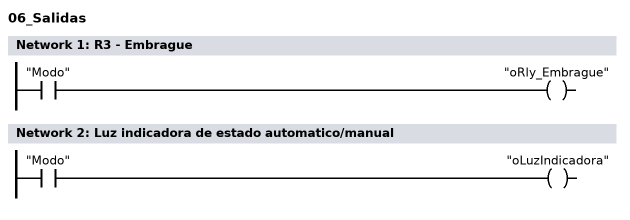
   RUNG wire#powerrail
      Contact( "Modo" )
      Coil( "oRly_Embrague" )
   END_RUNG
   // the same network as SCL:
   "oRly_Embrague" := "Modo";
END_REGION

REGION Network 2: Luz indicadora de estado automatico/manual
   RUNG wire#powerrail
      Contact( "Modo" )
      Coil( "oLuzIndicadora" )
   END_RUNG
   // the same network as SCL:
   "oLuzIndicadora" := "Modo";
END_REGION
END_FUNCTION

FUNCTION "02_Flancos" : Void   // FC6, LAD
{ S7_Optimized_Access := 'TRUE' }
VERSION : 0.1
   VAR_TEMP   // added for the SCL form of the ladder/FBD networks
      _w1 : Bool;
   END_VAR
BEGIN

REGION Network 1: Flanco Positivo Sensor Presencia de botella.
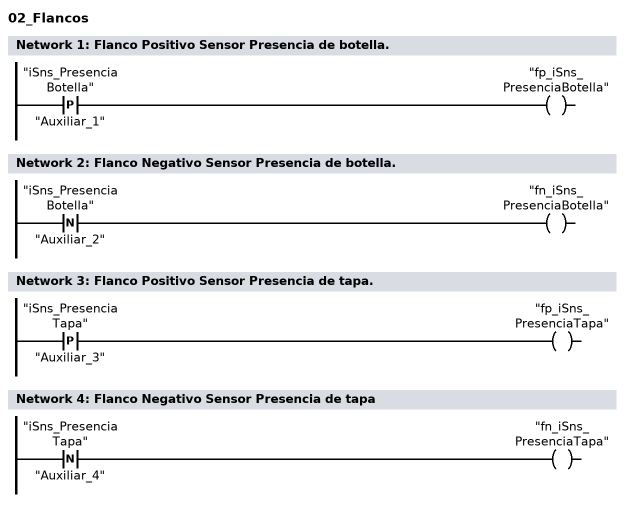
   RUNG wire#powerrail
      P_Contact(operand := "iSns_PresenciaBotella", bit := "Auxiliar_1")
      Coil( "fp_iSns_PresenciaBotella" )
   END_RUNG
   // the same network as SCL:
   #_w1 := "iSns_PresenciaBotella" AND NOT "Auxiliar_1";   // rising edge of "iSns_PresenciaBotella"
   "Auxiliar_1" := "iSns_PresenciaBotella";
   "fp_iSns_PresenciaBotella" := #_w1;
END_REGION

REGION Network 2: Flanco Negativo Sensor Presencia de botella.
   RUNG wire#powerrail
      N_Contact(operand := "iSns_PresenciaBotella", bit := "Auxiliar_2")
      Coil( "fn_iSns_PresenciaBotella" )
   END_RUNG
   // the same network as SCL:
   #_w1 := NOT "iSns_PresenciaBotella" AND "Auxiliar_2";   // falling edge of "iSns_PresenciaBotella"
   "Auxiliar_2" := "iSns_PresenciaBotella";
   "fn_iSns_PresenciaBotella" := #_w1;
END_REGION

REGION Network 3: Flanco Positivo Sensor Presencia de tapa.
   RUNG wire#powerrail
      P_Contact(operand := "iSns_PresenciaTapa", bit := "Auxiliar_3")
      Coil( "fp_iSns_PresenciaTapa" )
   END_RUNG
   // the same network as SCL:
   #_w1 := "iSns_PresenciaTapa" AND NOT "Auxiliar_3";   // rising edge of "iSns_PresenciaTapa"
   "Auxiliar_3" := "iSns_PresenciaTapa";
   "fp_iSns_PresenciaTapa" := #_w1;
END_REGION

REGION Network 4: Flanco Negativo Sensor Presencia de tapa
   RUNG wire#powerrail
      N_Contact(operand := "iSns_PresenciaTapa", bit := "Auxiliar_4")
      Coil( "fn_iSns_PresenciaTapa" )
   END_RUNG
   // the same network as SCL:
   #_w1 := NOT "iSns_PresenciaTapa" AND "Auxiliar_4";   // falling edge of "iSns_PresenciaTapa"
   "Auxiliar_4" := "iSns_PresenciaTapa";
   "fn_iSns_PresenciaTapa" := #_w1;
END_REGION
END_FUNCTION

FUNCTION "10_Simulacion" : Void   // FC7, LAD
{ S7_Optimized_Access := 'TRUE' }
VERSION : 0.1
   VAR_TEMP   // added for the SCL form of the ladder/FBD networks
      _w1 : Bool;
   END_VAR
BEGIN

REGION Network 1: Pulsador Inicio en caja mecanica.
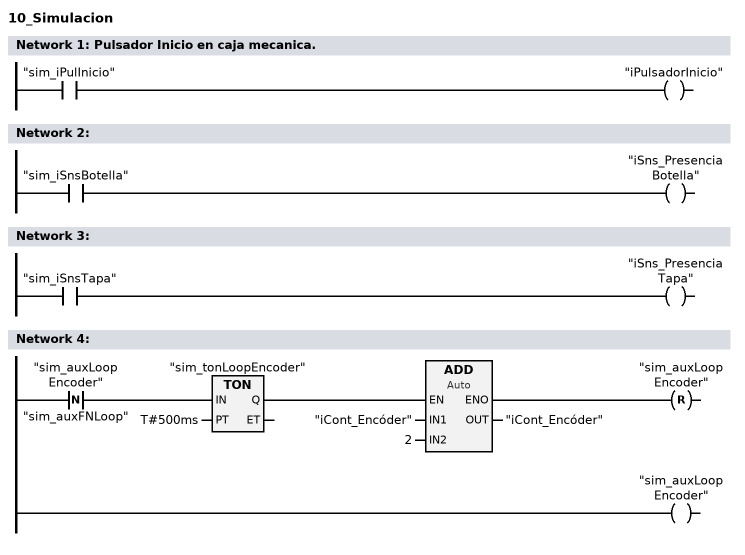
   RUNG wire#powerrail
      Contact( "sim_iPulInicio" )
      Coil( "iPulsadorInicio" )
   END_RUNG
   // the same network as SCL:
   "iPulsadorInicio" := "sim_iPulInicio";
END_REGION

REGION Network 2
   RUNG wire#powerrail
      Contact( "sim_iSnsBotella" )
      Coil( "iSns_PresenciaBotella" )
   END_RUNG
   // the same network as SCL:
   "iSns_PresenciaBotella" := "sim_iSnsBotella";
END_REGION

REGION Network 3
   RUNG wire#powerrail
      Contact( "sim_iSnsTapa" )
      Coil( "iSns_PresenciaTapa" )
   END_RUNG
   // the same network as SCL:
   "iSns_PresenciaTapa" := "sim_iSnsTapa";
END_REGION

REGION Network 4
   // ENO of a box is taken as its EN; it also drops when the box reports an error
   #_w1 := NOT "sim_auxLoopEncoder" AND "sim_auxFNLoop";   // falling edge of "sim_auxLoopEncoder"
   "sim_auxFNLoop" := "sim_auxLoopEncoder";
   "sim_tonLoopEncoder".TON(IN := #_w1, PT := T#500ms);
   IF "sim_tonLoopEncoder".Q THEN
       "iCont_Encóder" := "iCont_Encóder" + 2;
       "sim_auxLoopEncoder" := FALSE;
   END_IF;
   "sim_auxLoopEncoder" := TRUE;
END_REGION
END_FUNCTION

FUNCTION "07_HMI" : Void   // FC9, LAD
{ S7_Optimized_Access := 'TRUE' }
VERSION : 0.1
BEGIN

REGION Network 1
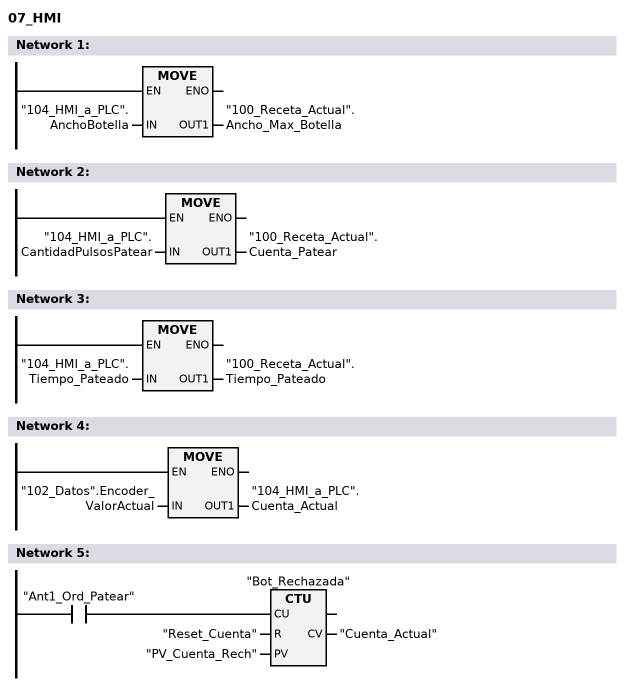
   RUNG wire#powerrail
      { S7_GenerateENO := "TRUE" } Move(in := "104_HMI_a_PLC".AnchoBotella, out1 => "100_Receta_Actual".Ancho_Max_Botella)
   END_RUNG
   // the same network as SCL:
   "100_Receta_Actual".Ancho_Max_Botella := "104_HMI_a_PLC".AnchoBotella;
END_REGION

REGION Network 2
   RUNG wire#powerrail
      { S7_GenerateENO := "TRUE" } Move(in := "104_HMI_a_PLC".CantidadPulsosPatear, out1 => "100_Receta_Actual".Cuenta_Patear)
   END_RUNG
   // the same network as SCL:
   "100_Receta_Actual".Cuenta_Patear := "104_HMI_a_PLC".CantidadPulsosPatear;
END_REGION

REGION Network 3
   RUNG wire#powerrail
      { S7_GenerateENO := "TRUE" } Move(in := "104_HMI_a_PLC".Tiempo_Pateado, out1 => "100_Receta_Actual".Tiempo_Pateado)
   END_RUNG
   // the same network as SCL:
   "100_Receta_Actual".Tiempo_Pateado := "104_HMI_a_PLC".Tiempo_Pateado;
END_REGION

REGION Network 4
   RUNG wire#powerrail
      { S7_GenerateENO := "TRUE" } Move(in := "102_Datos".Encoder_ValorActual, out1 => "104_HMI_a_PLC".Cuenta_Actual)
   END_RUNG
   // the same network as SCL:
   "104_HMI_a_PLC".Cuenta_Actual := "102_Datos".Encoder_ValorActual;
END_REGION

REGION Network 5
   "Bot_Rechazada".CTU(CU := "Ant1_Ord_Patear",
                       R := "Reset_Cuenta",
                       PV := "PV_Cuenta_Rech",
                       CV => "Cuenta_Actual");
END_REGION
END_FUNCTION

ORGANIZATION_BLOCK "Main"   // OB1, LAD, ProgramCycle
TITLE = "Main Program Sweep (Cycle)"
{ S7_Optimized_Access := 'TRUE' }
VERSION : 0.1
BEGIN

REGION Network 1
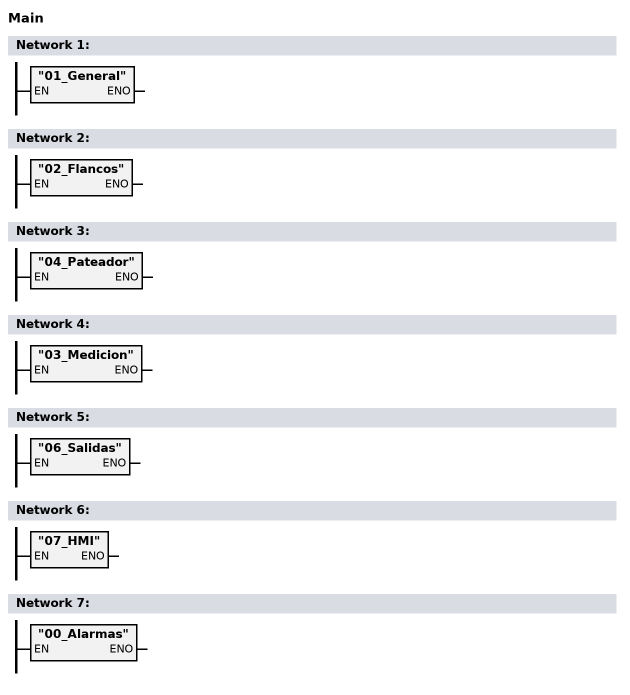
   RUNG wire#powerrail
      "01_General"()
   END_RUNG
   // the same network as SCL:
   "01_General"();
END_REGION

REGION Network 2
   RUNG wire#powerrail
      "02_Flancos"()
   END_RUNG
   // the same network as SCL:
   "02_Flancos"();
END_REGION

REGION Network 3
   RUNG wire#powerrail
      "04_Pateador"()
   END_RUNG
   // the same network as SCL:
   "04_Pateador"();
END_REGION

REGION Network 4
   RUNG wire#powerrail
      "03_Medicion"()
   END_RUNG
   // the same network as SCL:
   "03_Medicion"();
END_REGION

REGION Network 5
   RUNG wire#powerrail
      "06_Salidas"()
   END_RUNG
   // the same network as SCL:
   "06_Salidas"();
END_REGION

REGION Network 6
   RUNG wire#powerrail
      "07_HMI"()
   END_RUNG
   // the same network as SCL:
   "07_HMI"();
END_REGION

REGION Network 7
   RUNG wire#powerrail
      "00_Alarmas"()
   END_RUNG
   // the same network as SCL:
   "00_Alarmas"();
END_REGION
END_ORGANIZATION_BLOCK

ORGANIZATION_BLOCK "Inicializacion"   // OB100, LAD, Startup
TITLE = Inicializacion / "Complete Restart"
{ S7_Optimized_Access := 'TRUE' }
VERSION : 0.1
// En este bloque inicializamos todas las varibles que necesitan inicializacion
   VAR_INPUT
      LostRetentive : Bool;   // True if retentive data are lost
      LostRTC : Bool;   // True if date and time are lost
   END_VAR
BEGIN

REGION Network 1: Este Bit Siempre está en 0
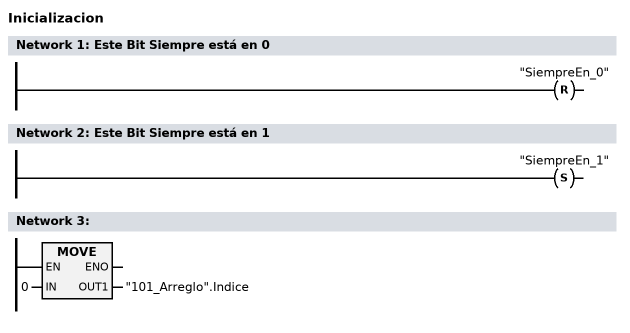
   RUNG wire#powerrail
      R_Coil( "SiempreEn_0" )
   END_RUNG
   // the same network as SCL:
   "SiempreEn_0" := FALSE;
END_REGION

REGION Network 2: Este Bit Siempre está en 1
   RUNG wire#powerrail
      S_Coil( "SiempreEn_1" )
   END_RUNG
   // the same network as SCL:
   "SiempreEn_1" := TRUE;
END_REGION

REGION Network 3
   RUNG wire#powerrail
      { S7_GenerateENO := "TRUE" } Move(in := 0, out1 => "101_Arreglo".Indice)
   END_RUNG
   // the same network as SCL:
   "101_Arreglo".Indice := 0;
END_REGION
END_ORGANIZATION_BLOCK

(* ===== HMI "HMI_RT_2" =====
system functions are stored by id; their names below are inferred from use
connection "Conexión_2": ETHERNET, SMART_S7_1200_OMS
connection "HMI_Conexión_1": ETHERNET, SMART_S7_1200_OMS

HMI tags "Tabla de variables estándar"
   "104_HMI_a_PLC_Reset" : Bool = PLC "104_HMI_a_PLC".Reset, 1 s
   "AnchoBotella" : DInt = PLC "104_HMI_a_PLC".AnchoBotella AT %DB1.DBX0.0, 1 s
   "CantidadPulsosPatear" : DInt = PLC "104_HMI_a_PLC".CantidadPulsosPatear AT %DB1.DBX0.0, 1 s
   "Tiempo_Pateado" : Time = PLC "104_HMI_a_PLC".Tiempo_Pateado AT %DB1.DBX0.0, 1 s
   "Cuenta_Actual_encoder" : DInt = PLC "104_HMI_a_PLC".Cuenta_Actual AT %DB1.DBD0, 1 s
   "Reset_Cuenta" : Bool = PLC Reset_Cuenta AT %M3.0, 1 s
   "Cuenta_Actual_Recha" : Int = PLC Cuenta_Actual AT %MW12, 1 s

HMI tags "01_ALARMAS"
   "ALARMAS_1" : Word AT %DB71.DBW0, 1 s
   "ALARMAS_2" : Word AT %DB71.DBW2, 1 s

discrete alarms
   1: 'Parada manual accionada.', class Errors, trigger "ALARMAS_1" bit 0
   2: 'Se detectó sobreesfuerzo en los dedos del pateador.', class Errors, trigger "ALARMAS_1" bit 1
   3: 'Falla en encoder_ no cuenta entre dos botellas', class Errors, trigger "ALARMAS_1" bit 2
   4: 'Falla por cantidad de cuentas', class Errors, trigger "ALARMAS_1" bit 3
   5: 'Se supero la máxima cantidad de botellas rechazadas permitidas', class Errors, trigger "ALARMAS_1" bit 4
   6: '', class Errors, trigger "ALARMAS_1" bit 5
   7: '', class Errors, trigger "ALARMAS_1" bit 6
   8: '', class Errors, trigger "ALARMAS_1" bit 7
   9: '', class Errors, trigger "ALARMAS_1" bit 8
   10: '', class Errors, trigger "ALARMAS_1" bit 9
   11: '', class Errors, trigger "ALARMAS_1" bit 10
   12: '', class Errors, trigger "ALARMAS_1" bit 11
   13: '', class Errors, trigger "ALARMAS_1" bit 12
   14: '', class Errors, trigger "ALARMAS_1" bit 13
   15: '', class Errors, trigger "ALARMAS_1" bit 14
   16: '', class Errors, trigger "ALARMAS_1" bit 15
   17: '', class Errors, trigger "ALARMAS_2" bit 0
   18: '', class Errors, trigger "ALARMAS_2" bit 1
   19: '', class Errors, trigger "ALARMAS_2" bit 2
   20: '', class Errors, trigger "ALARMAS_2" bit 3
   21: '', class Errors, trigger "ALARMAS_2" bit 4
   22: '', class Errors, trigger "ALARMAS_2" bit 5
   23: '', class Errors, trigger "ALARMAS_2" bit 6
   24: '', class Errors, trigger "ALARMAS_2" bit 7
   25: '', class Errors, trigger "ALARMAS_2" bit 8
   26: '', class Errors, trigger "ALARMAS_2" bit 9
   27: '', class Errors, trigger "ALARMAS_2" bit 10
   28: '', class Errors, trigger "ALARMAS_2" bit 11
   29: '', class Errors, trigger "ALARMAS_2" bit 12
   30: '', class Errors, trigger "ALARMAS_2" bit 13
   31: '', class Errors, trigger "ALARMAS_2" bit 14
   32: '', class Errors, trigger "ALARMAS_2" bit 15

text list "Imagen Seleccionada": 1 'Imagen Principal'; 2 'Config Tiro Grupo 1'; 3 'Config Tiro Grupo 2'; 4 'Bob 1 de Grupo 1'; 5 'Bob 2 de Grupo 1'; 6 'Bob 1 de Grupo 2'; 7 'Bob 2 de Grupo 2'; 8 'Alarmas'; 9 'Historial'; 10 'Recetas'

text list "Error Configuracion Puerto Modbus": 33152 'Valor no válido para la ID de puerto (dirección errónea del módulo de comunicación).'; 33153 'Valor no válido para la velocidad de transferencia.'; 33154 'Valor no válido para la paridad.'; 33155 'Valor no válido para el tiempo excedido de la respuesta (el lapso de tiempo hasta que se comunica el tiempo excedido debe ser como mínimo 25 ms).'; 33156 'Puntero incorrecto en el parámetro MB_DB hacia el DB de instancia de la instrucción "MB_MASTER" o "MB_SLAVE".'

text list "Error Comunicación Modbus": 32968 'Timeout del esclavo. Compruebe la velocidad de transferencia, la paridad y las conexiones del esclavo.'; 32977 'El receptor ha solicitado un control de flujo para interrumpir una transmisión en curso, pero la transmisión no se ha vuelto a activar en el tiempo de espera. Este error también se crea en el control de flujo por hardware cuando el receptor no detecta ningún CTS en el tiempo de espera.'; 32978 'La solicitud de transmisión se ha cancelado, porque no se recibe ninguna señal DSR del DCE.'; 32992 'El aviso se ha finalizado porque el búfer de recepción está lleno.'; 32993 'El aviso se ha finalizado por un error de paridad.'; 32994 'El aviso se ha finalizado por un error de telegrama.'; 32995 'El aviso se ha finalizado por un error de desbordamiento.'; 32996 'El aviso se ha cancelado, porque la longitud indicada excede el tamaño del búfer total.'; 33152 'Valor no válido para la ID de puerto.'; 33158 'Dirección de estación Modbus no válida'; 33160 'Valor no válido en el parámetro MODE para una llamada de difusión general.'; 33161 'Valor no válido para la dirección de datos.'; 33162 'Valor no válido para la longitud de datos.'; 33163 'Puntero no válido hacia el origen o destino de datos local: tamaño incorrecto'; 33164 'Puntero no válido en el parámetro DATA_PTR. Utilice un puntero hacia un área de marcas o un DB con el tipo de acceso "Estándar: compatible con S7-300/400".'; 33280 'El puerto está ocupado procesando una solicitud de transmisión'; 33664 'Error CRC.'; 33665 'Código de función no soportado.'; 33666 'Error en la longitud de datos.'; 33667 'Error en la dirección de los datos o dirección fuera del rango válido de DATA_PTR.'; 33668 'Error en el valor de datos.'; 33669 'Valor del código de diagnóstico de datos no soportado (código de función 08).'; 33670 'El código de función de la respuesta no concuerda con el código de función de la consulta.'; 33671 'Respuesta de un esclavo equivocado.'; 33672 'La respuesta del esclavo a una llamada de escritura no es correcta. Los datos enviados por el esclavo no concuerdan con la consulta del maestro.'

text list "Fallas_V90": 1000 'F1000: Error SW interno'; 1001 'F1001: Excepción Floating-Point'; 1002 'F1002: Error SW interno'; 1003 'F1003: Retardo de acuse al acceder a memoria'; 1005 'F1015: Error SW interno'; 1008 'F1018: Arranque cancelado varias veces'; 1030 'F1030: Pérdida de signo de actividad para control maestro'; 1611 'F1611: SI CU: Defecto detectado'; 1910 'F1910: Fieldbus: setpoint timeout'; 7011 'F7011: Sobrecalentamiento del motor'; 7085 'F7085: Parámetros de control en lazo abierto/lazo cerrado'; 7093 'F7093: Accionamiento: Error de señal de prueba'; 7220 'F7220: Drive: Master control by PLC missing'; 7403 'F7403: Umbral inferior de tensión en circuito intermedio alcanzado'; 7404 'F7404: Umbral superior de tensión en circuito intermedio alcanzado'; 7410 'F7410: Salida de regulador de corriente limitada'; 7412 'F7412: Ángulo de conmutación erróneo (modelo de motor)'; 7420 'F7420: Accionamiento: Frecuencia propia filtro consigna intensidad > Frecuencia de Shannon'; 7430 'F7430: No es posible conmutar a funcionamiento controlado de par en lazo abierto'; 7431 'F7431: No es posible conmutar al modo sin encóder'; 7442 'F7442: RP: Multivuelta no compatible con el margen módulo'; 7443 'F7443: Coordenada del punto de referencia fuera del margen permitido'; 7450 'F7450: La vigilancia de parada ha respondido'; 7451 'F7451: La vigilancia de posición ha respondido'; 7452 'F7452: Error de seguimiento excesivo'; 7453 'F7453: Error de acondicionamiento de valor real de posición'; 7454 'F7458: PosS: Levas de referencia no encontradas'; 7459 'F7459: No existe marca cero'; 7460 'F7460: PosS: Fin de leva de referencia no encontrado'; 7464 'F7464: PosS: El bloque de desplazamiento es incoherente'; 7475 'F7475: PosS: Posición de destino < Inicio de margen de desplazamiento'; 7476 'F7476: PosS: Posición de destino > Fin de margen de desplazamiento'; 7481 'F7481: PosS: Posición de eje < Final de carrera de software Menos'; 7482 'F7482: PosS: Posición de eje > Final de carrera de software Más'; 7490 'F7490: Señal de habilitación anulada durante desplazamiento'; 7491 'F7491: Leva de parada Menos alcanzada'; 7492 'F7492: Leva de parada Más alcanzada'; 7493 'F7493: RP: Desbordamiento del rango de valores para la posición real'; 7599 'F7599: Encóder 1: el ajuste no es posible'; 7800 'F7800: Accionamiento: No hay etapa de potencia.'; 7801 'F7801: Sobrecorriente del motor'; 7802 'F7802: Alimentación o etapa de potencia no lista'; 7815 'F7815: Se ha modificado la etapa de potencia'; 7900 'F7900: Motor bloqueado/Regulador de velocidad en tope'; 7901 'F7901: Sobrevelocidad del motor'; 7995 'F7995: Fallo de identificación del motor'; 30001 'F30001: Etapa de potencia: Sobrecorriente'; 30002 'F30002: Sobretensión en circuito intermedio'; 30003 'F30003: Subtensión en circuito intermedio'; 30004 'F30004: Sobretemperatura en disipador de convertidor'; 30005 'F30005: Etapa de potencia: Sobrecarga I2t'; 30011 'F30011: Pérdida de fase de red en el circuito principal'; 30015 'F30015: Pérdida de fase del cable del motor'; 30021 'F30021: Defecto a tierra'; 30027 'F30027: Vigilancia de tiempo de circuito intermedio en precarga'; 30036 'F30036: Sobretemperatura en interior'; 30050 'F30050: Sobretensión de alimentación de 24 V'; 31100 'F31100: Error cero en distancia entre marcas'; 31101 'F31101: Marca cero fallida'; 31110 'F31110: Comunicación serie con perturbaciones'; 31112 'F31112: Bit de error ajustado en protocolo serie'; 31117 'F31117: Señales de error de inversión A/B/R'; 31130 'F31130: Marca cero y posición de sincronización aprox. incorrectas'; 31150 'F31150: Error de inicialización'; 52903 'F52903: Error de incoherencia entre el estado de fallo y la memoria de fallos'; 52904 'F52904: Cambio del modo de control'; 52911 'F52911: Error de valor para la limitación de par positivo'; 52912 'F52912: Error de valor para la limitación de par negativo'; 52931 'F52931: Límite del reductor'; 52933 'F52933: Límite del reductor PTO'; 52980 'F52980: Motor de encóder absoluto sustituido'; 52981 'F52981: Discrepancia con motor de encóder absoluto'; 52983 'F52983: Ningún encóder detectado'; 52984 'F52984: Motor de encóder incremental no configurado'; 52985 'F52985: Motor de encóder absoluto erróneo'; 52987 'F52987: Encóder absoluto sustituido'; 52988 'Error. No se puede determinar el tipo de falla'

text list "Alarmas_90": 1009 'A1009: Control Unit Sobretemperatura'; 1019 'A1019: Fallo al escribir en el cartucho intercambiable'; 1032 'A1032: Almacenamiento necesario de todos los parámetros'; 1045 'A1045: Datos de configuración no válidos'; 1920 'A1920: Bus en accionamiento: Recibir consignas tras To'; 1932 'A1932: Falta sincronización de ciclo del bus en accionamiento para DSC'; 5000 'A5000: Sobretemperatura en disipador de convertidor'; 7012 'A7012: Modelo de temperatura del motor 1/3 Exceso de temperatura'; 7441 'A7441: RP: Guardar offset de posición de la calibración del encóder absoluto'; 7456 'A7456: PosS: Velocidad de consigna limitada'; 7461 'A7461: PosS: Punto de referencia no ajustado'; 7469 'A7469: PosS: Bloque de desplazamiento Posición de destino < Final de carrera software Menos'; 7470 'A7470: PosS: Bloque de desplazamiento Posición de destino > Final de carrera software Más'; 7471 'A7471: PosS: Bloque de desplazamiento Posición de destino fuera del margen módulo'; 7472 'A7472: PosS: Bloque de desplazamiento ABS_POS/ABS_NEG imposible'; 7473 'A7473: PosS: Inicio de margen de desplazamiento alcanzado'; 7474 'A7474: PosS: Fin de margen de desplazamiento alcanzado'; 7477 'A7477: PosS: Posición de destino < Final de carrera software Menos'; 7478 'A7478: PosS: Posición de destino > Final de carrera software Más'; 7479 'A7479: PosS: Final de carrera software Menos alcanzado'; 7480 'A7480: PosS: Final de carrera software Más alcanzado'; 7496 'A7496: Falta habilitación SON'; 7576 'A7576: Modo sin encóder activo debido a un fallo'; 7582 'A7582: Error de acondicionamiento de valor real de posición'; 7585 'A7585: P-TRG o CLR activo'; 7805 'A7805: Sobrecarga I2t de la etapa de potencia'; 7965 'A7965: Necesario guardar'; 7971 'A7971: Offset de ángulo de conmutación Determinación activada'; 7991 'A7991: Identificación de datos de motor activada'; 30016 'A30016: Alimentación de carga desconectada'; 30031 'A30031: Limitación de intensidad por hardware en la fase U'; 31411 'A31411: Encóder absoluto señaliza alarmas internas'; 31412 'A31412: Bit de error ajustado en protocolo serie'; 52900 'A52900: Fallo al copiar datos'; 52901 'A52901: La resistencia de frenado alcanza el umbral de alarma'; 52902 'A52902: Emergencia desconectada'; 52932 'A52932: Límite máx. PTO'

screen "01_Alarmas" 320x240, template "Plantilla_Principal"
   AlarmView "Visor de avisos_1" at 0,32 size 319x177
   Button "Botón_1" at 265,209 size 54x30; TextOff 'Reset Alarmas'
      on Release: ResetBit("104_HMI_a_PLC_Reset")
      on Press: SetBit("104_HMI_a_PLC_Reset")
   Softkey "Softkey_F6" at 266,202 size 53x38
      on KeyUp: ResetBit("104_HMI_a_PLC_Reset")
      on KeyDown: SetBit("104_HMI_a_PLC_Reset")

screen "09_Hitorial_anulado" 320x240, template "Plantilla_Principal"
   AlarmView "Visor de avisos_1" at 0,32 size 319x177

screen "Inicio" 320x240, template "Plantilla_Principal"
   TextField "Campo de texto_1" at 13,36 size 89x13; Text 'Ancho de Botella:'
   TextField "Campo de texto_2" at 13,65 size 174x13; Text 'Cantidad de Pulsos para Rechazar:'
   TextField "Campo de texto_3" at 13,94 size 101x13; Text 'Tiempo de Pateado:'
   IOField "Campo ES_1" at 221,31 size 70x23; FormatPattern 9999; Unit  ctas
      ProcessValue <- "AnchoBotella"
   IOField "Campo ES_2" at 221,60 size 70x23; FormatPattern 9999; Unit  ctas
      ProcessValue <- "CantidadPulsosPatear"
   IOField "Campo ES_3" at 221,89 size 70x23; FormatPattern 9999; Unit  ms
      ProcessValue <- "Tiempo_Pateado"
   TextField "Campo de texto_4" at 13,124 size 130x13; Text 'Valor actual de encoder:'
   IOField "Campo ES_4" at 202,119 size 89x23; FormatPattern 99999999; Unit  ctas
      ProcessValue <- "Cuenta_Actual_encoder"
   TextField "Campo de texto_5" at 13,154 size 136x13; Text 'Cant. Botellas Rechazadas:'
   IOField "Campo ES_5" at 221,149 size 70x23; FormatPattern 99999; Unit  Bot
      ProcessValue <- "Cuenta_Actual_Recha"
   Button "Botón_1" at 214,210 size 51x29; TextOff 'Reset cuenta'
      on Release: ResetBit("Reset_Cuenta")
      on Press: SetBit("Reset_Cuenta")

Template "Plantilla_Principal" 320x240
   SymbolicIOField "Imagen_campo_ES_simbólico_1" at 40,1 size 280x16; TextOn '1'; TextOff '0'
      on Change: ActivateScreenByNumber("HMI_a_PLC_NroImagenActual", 0)
   Button "Template_Button_4" at 54,209 size 52x30; TextOff 'Text'
   DateTimeField "HmiScreenItemData_1" at 243,1 size 77x16
   Button "Template_Button_5" at 1,209 size 52x30; TextOn 'NavigateHome'; TextOff 'NavigateHome'; PictureOn "NavigateHome_KTP600_Basic_PN"; PictureOff "NavigateHome_KTP600_Basic_PN"
      on Release: ActivateScreen("Inicio", 0)
   Button "Template_Button_6" at 266,209 size 52x30; TextOff 'Alarmas'
      on Release: ActivateScreen("01_Alarmas", 0)
   Button "Template_Button_1" at 107,209 size 52x30; TextOff 'Text'
   Button "Template_Button_2" at 160,209 size 52x30; TextOff 'Text'
   TextField "Plantilla_Campo de texto_1" at 48,2 size 186x14; Text 'Rechazador Stork 3'
   GraphicView "Plantilla_Visor de gráficos_1" at 0,1 size 41x16; Picture "eProC logo Gris B"
   Button "Template_Button_3" at 213,209 size 52x30; TextOff 'Text'
   Softkey "Softkey_F6" at 266,202 size 53x38
      on KeyUp: ActivateScreen("01_Alarmas", 3)
   Softkey "Softkey_F1" at 1,202 size 53x38
      on KeyUp: ActivateScreen("Inicio", 0)
*)